// TIA Portal V20 export
DATA_BLOCK "CallEquipment_DB"   // DB114
{ DB_Accessible_From_OPC_UA := 'FALSE' }
// stored: AssignedProDiagFB Unit1.Em12.ProDiag, DBAccessibleFromOPCUA false, DBAccessibleFromWebserver false, InstanceOfName Unit1.Em12.CallEquipment, InstanceOfType FB, Namespace Unit1.Em12
"Unit1.Em12.CallEquipment"
   // VAR_INPUT
   //    ZoneOperationEnable { ExternalWritable := 'False'} : "LWONIK_typeSafetyZoneManualOperation";
   // END_VAR
   // VAR_IN_OUT
   //    unitStatus : "LAF_typeUnitStatus";
   //    emFeedback : "LUC_typeEmFeedback";
   //    unitAlarmDB : "LAF_typeAlarms";
   // END_VAR
   // VAR
   //    InstStackNgBoxSequence { ExternalWritable := 'False'} : "Unit1.Em12.Sequence_1_StackNgBox";
   //    instStackNgBoxHomeJob1 { ExternalWritable := 'False'} : "LAF_SelectJob";
   //    instStackNgBoxLoadJob2 { ExternalWritable := 'False'} : "LAF_SelectJob";
   //    instStackNgBoxUnloadJob3 { ExternalWritable := 'False'} : "LAF_SelectJob";
   //    instCmStackNgBoxFullDetect { ExternalWritable := 'False'} : "LBC_DigitalSignalCn";
   //    instCmStackNgBoxDetect { ExternalWritable := 'False'} : "LBC_DigitalSignalCn";
   //    instCmStackNgBoxLoadingUpDown { ExternalWritable := 'False'} : "LBC_TwoWayActuatorCn";
   //    instCmStackNgBoxUnitMoverBwdFwd { ExternalWritable := 'False'} : "LBC_TwoWayActuatorCn";
   //    instCmStackNgBoxClampLeftOpenClose { ExternalWritable := 'False'} : "LBC_TwoWayActuatorCn";
   //    instCmStackNgBoxClampRightOpenClose { ExternalWritable := 'False'} : "LBC_TwoWayActuatorCn";
   //    instCmStackNgBoxClampMoverOpenClose { ExternalWritable := 'False'} : "LBC_TwoWayActuatorCn";
   //    instCmStackNgBoxLiftDownUp { ExternalWritable := 'False'} : "LBC_TwoWayActuatorCn";
   //    instCmStackNgBoxLockDownUp { ExternalWritable := 'False'} : "LBC_TwoWayActuatorCn";
   //    instManageAlarms { ExternalWritable := 'False'} : "LAF_ManageAlarms";
   //    instEventsPFE { ExternalWritable := 'False'} : "Unit1.Em12.EventsPFE";
   //    statUnitStatus { ExternalWritable := 'False'} : "LAF_typeUnitStatus";
   //    statPartData { ExternalWritable := 'False'} : "LER_typePartData";
   //    statTonTime { ExternalWritable := 'False'} : Array[0..999] of TON_TIME;
   //    statTofTime { ExternalWritable := 'False'} : Array[0..99] of TOF_TIME;
   //    statPulse { ExternalWritable := 'False'} : Array[0..999] of Bool;
   //    statEnableManualCmds { ExternalWritable := 'False'} : Bool;
   //    "*** Interlock TwoWay ***" { S7_SetPoint := 'True'} : "LER_Axis_Homing";
   //    instCmStackNgBoxLoadingUpDownInterlock { S7_SetPoint := 'True'} : Array[0..2] of "LER_Actuator";
   //    instCmStackNgBoxUnitMoverBwdFwdInterlock { S7_SetPoint := 'True'} : Array[0..2] of "LER_Actuator";
   //    instCmStackNgBoxClampLeftOpenCloseInterlock { S7_SetPoint := 'True'} : Array[0..2] of "LER_Actuator";
   //    instCmStackNgBoxClampRightOpenCloseInterlock { S7_SetPoint := 'True'} : Array[0..2] of "LER_Actuator";
   //    instCmStackNgBoxClampMoverOpenCloseInterlock { S7_SetPoint := 'True'} : Array[0..2] of "LER_Actuator";
   //    instCmStackNgBoxLiftDownUpInterlock { S7_SetPoint := 'True'} : Array[0..2] of "LER_Actuator";
   //    instCmStackNgBoxLockDownUpInterlock { S7_SetPoint := 'True'} : Array[0..2] of "LER_Actuator";
   //    StackNgBoxLoadingUpDown_Inpos : Array[0..2] of Struct
   //       "Int" : Array[1..10] of Bool;
   //    END_STRUCT;
   //    StackNgBoxUnitMoverBwdFwd_Inpos : Array[0..2] of Struct
   //       "Int" : Array[1..10] of Bool;
   //    END_STRUCT;
   //    StackNgBoxClampLeftOpenClose_Inpos : Array[0..2] of Struct
   //       "Int" : Array[1..10] of Bool;
   //    END_STRUCT;
   //    StackNgBoxClampRightOpenClose_Inpos : Array[0..2] of Struct
   //       "Int" : Array[1..10] of Bool;
   //    END_STRUCT;
   //    StackNgBoxClampMoverOpenClose_Inpos : Array[0..2] of Struct
   //       "Int" : Array[1..10] of Bool;
   //    END_STRUCT;
   //    StackNgBoxLiftDownUp_Inpos : Array[0..2] of Struct
   //       "Int" : Array[1..10] of Bool;
   //    END_STRUCT;
   //    StackNgBoxLockDownUp_Inpos : Array[0..2] of Struct
   //       "Int" : Array[1..10] of Bool;
   //    END_STRUCT;
   //    citi_Ptrig : Array[0..20] of Bool;
   //    citiTon : Array[0..20] of TON_TIME;
   //    citi : Time;
   //    citiTest : Array[0..20] of Bool;
   // END_VAR
BEGIN
END_DATA_BLOCK
